DATA_BLOCK "DB_General_Status"
TITLE =%version: 0.05 % CN: 20
//History:
//This version  %created_by: nlhdl %
//              %date_created: maandag 7 december 2015 15:56:08 %
//              %release: VI_RAW/RA_Dev %
//
//Modification History:                                   By:    Date:     Rev:
//----------------------------------------------------  -------  --------  -----
//ra#9751: Add source files ECS-P to VI_RAW             nlHdL    14-12-15   0.05
//ra#9751: Add source files ECS-P to VI_RAW             nlHdL    07-12-15   0.05
//7324: ECS-P General from the RD to RA for platform    nlHdL    06-07-15   0.05
//20643: DB moved to NON RETAIN memory                  nlHdL    16-09-14   0.05
//15797: Keyword release added                          nlwwij   26-09-13   0.04
//CR7631 Insert key word for code generator             nlple    06-10-11   0.03
//Updated version numbers                               nlMRe    15-09-10   0.02
//Initial revision                                      nlRSwi   03-09-10   1
//
FAMILY : General
VERSION : 0.0
NON_RETAIN


  STRUCT
   Insert : INT ;	// Insertion point for the S7 Code Generator
  END_STRUCT ;
BEGIN
END_DATA_BLOCK
